// TIA Portal V18 export
ORGANIZATION_BLOCK "Cyclic interrupt"   // OB31, FBD, CyclicInterrupt
{ S7_Optimized_Access := 'TRUE' }
VERSION : 0.1
// stored: AutoNumber true, IsIECCheckEnabled false, SetENOAutomatically false
   VAR_INPUT
      Initial_Call : Bool;   // Initial call of this OB
      Event_Count : Int;   // Events discarded
   END_VAR
BEGIN

REGION Network 1
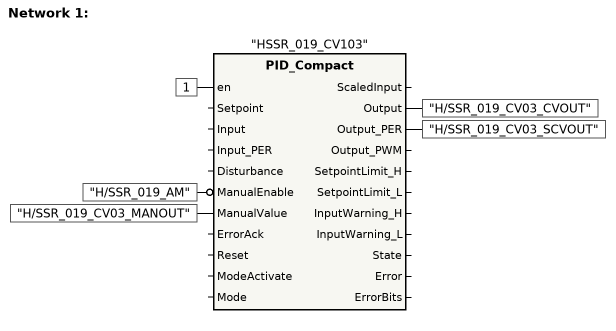
   IF 1 THEN
       "HSSR_019_CV103"(ManualEnable := NOT "H/SSR_019_AM",   // PID_Compact
                        ManualValue := "H/SSR_019_CV03_MANOUT",
                        Output => "H/SSR_019_CV03_CVOUT",
                        Output_PER => "H/SSR_019_CV03_SCVOUT");
   END_IF;
END_REGION
END_ORGANIZATION_BLOCK
